// TIA Portal V19 export
VAR_GLOBAL   // PLC tag table "Unit_DefaultTagTable_2"
END_VAR
